FUNCTION_BLOCK FB_Test
VAR_INPUT
END_VAR
VAR_OUTPUT
END_VAR
VAR
	fbEvent: 			Tc3_Event.FB_Event;
	bVerbose:			BOOL;
	bInfo:				BOOL;
	bWarning:			BOOL;
	bError:				BOOL;
	bCritical:			BOOL;

END_VAR


	
	fbEvent();
	
	IF bVerbose THEN
		fbEvent.P_Argument.M_AddINT(134052566194980000);
		fbEvent.P_Argument.M_AddSTRING('mm');
		fbEvent.M_Verbose('V message %s %s');
	END_IF
	
	IF bInfo THEN
		fbEvent.P_Argument.M_AddREAL(33.134581234, 3);
		fbEvent.P_Argument.M_AddSTRING('mm');
		fbEvent.M_Info(828536003, 'I message %s %s');
	END_IF
	
	IF bWarning THEN
		fbEvent.M_Warning(475719253, 'W message');
		fbEvent.M_Warning(475719253, 'W message');
	END_IF
	
	IF bError THEN
		fbEvent.M_Error(475719235, 'E message');
	END_IF
	
	IF bCritical THEN
		fbEvent.M_Critical(0, 'C message'); ///839384782
	END_IF

PROPERTY PUBLIC P_Event : reference to FB_event
GET
P_Event ref= fbEvent;
END_GET
END_PROPERTY

END_FUNCTION_BLOCK

(* stored: Version 1.1.0.1
   POU FB_Test: Id {8cd1133b-3477-41c9-9026-b27d8cb7f6d2}, SpecialFunc None
   Property P_Event: Id {1b280b73-a5c7-4186-ac99-29403b5a1044}
   Get Get: Id {f7a9f415-12a5-443c-b0d8-84df15e2089b} *)
